SUBAPPLICATION IX_TO_logiBUS_LED_strip_QX (* Taster IX schaltet einen LED-Strip blinkend (Farbe, Frequenz, Strip-Nummer parametrierbar). Generisch. *)
  (* Standard: 61499-2 *)
  (* Version 1.0, 2026-09-09, Franz Höpfinger, Meisterschulen am Ostbahnhof, Ausgelagert aus Uebung_033_sub zur Wiederverwendung. *)
  PACKAGE MyLib::sys;
  IMPORT logiBUS::io::DI::logiBUS_DI_S;
  IMPORT logiBUS::io::DO_LED::LED_COLOURS;
  IMPORT logiBUS::io::DO_LED::LED_FREQ;
  IMPORT logiBUS::io::DI::logiBUS_DI::Invalid;
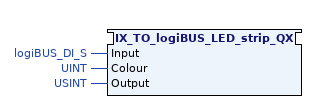
  VAR_INPUT
    Input : logiBUS::io::DI::logiBUS_DI_S := Invalid; (* Identify the Input Input_I1..I8 *)
    Colour : UINT := LED_COLOURS::LED_GREEN; (* This identify the Colour. *)
    Output : USINT; (* Identify the Output Number of Strip *)
  END_VAR
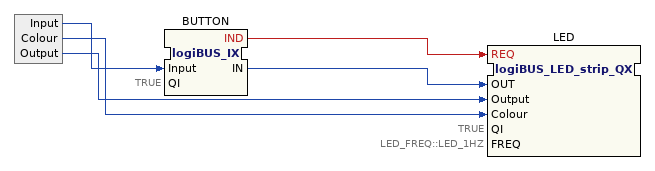
  FBS
    LED : logiBUS::io::DO_LED::logiBUS_LED_strip_QX(QI := TRUE, FREQ := LED_FREQ::LED_1HZ);
    BUTTON : logiBUS::io::DI::logiBUS_IX(QI := TRUE);
  END_FBS
  EVENT_CONNECTIONS
    BUTTON.IND TO LED.REQ;
  END_CONNECTIONS
  DATA_CONNECTIONS
    BUTTON.IN TO LED.OUT;
    Input TO BUTTON.Input;
    Output TO LED.Output;
    Colour TO LED.Colour;
  END_CONNECTIONS
END_SUBAPPLICATION
